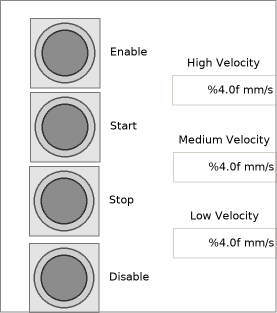
VISUALIZATION Controls_LD  // 277x313
    PushSwitchLed (30,18 70x70), variable: P_LD.MainCommands.Enable, behaviour: TOGGLE, style: Switch-PushSwitchLed-Gray
    Label (107,37 75x30), "Enable"
    Label (107,111 75x30), "Start"
    PushSwitchLed (30,92 70x70), variable: P_LD.MainCommands.Start, behaviour: TOGGLE, style: Switch-PushSwitchLed-Gray
    Label (106,185 75x30), "Stop"
    PushSwitchLed (29,166 70x70), variable: P_LD.MainCommands.Stop, behaviour: TOGGLE, style: Switch-PushSwitchLed-Gray
    Label (106,262 75x30), "Disable"
    PushSwitchLed (29,243 70x70), variable: P_LD.MainCommands.Disable, behaviour: TOGGLE, style: Switch-PushSwitchLed-Gray
    Textfield (172,75 104x30), "%4.0f mm/s", text variable: P_LD.highVelocity
        OnMouseClick: write the text variable via VisuDialogs.Numpad, min 1, max 2000, format %f.0
    Label (175,54 97x18), "High Velocity"
    Textfield (173,152 104x30), "%4.0f mm/s", text variable: P_LD.mediumVelocity
        OnMouseClick: write the text variable via VisuDialogs.Numpad, min 1, max 2000, format %f.0
    Label (176,131 97x18), "Medium Velocity"
    Textfield (173,228 104x30), "%4.0f mm/s", text variable: P_LD.lowVelocity
        OnMouseClick: write the text variable via VisuDialogs.Numpad, min 1, max 2000, format %f.0
    Label (176,207 97x18), "Low Velocity"
END_VISUALIZATION

(* stored: Version 1.1.0.1
   Visu Controls_LD: Id {716113f3-45a7-47d0-95b2-7a271b6a8622} *)
